FUNCTION_BLOCK PUBLIC LotLogging
VAR_INPUT
END_VAR
VAR_OUTPUT
END_VAR
VAR
	PrevLotInProgress : BOOL;
	TimeToLogLot : TON;
END_VAR

IF (NOT LotsData.Lot.LotInProgress) AND PrevLotInProgress THEN
	// create a lot report here and store it
	P_TextModeWriteLot.WriteData := TRUE;	   
END_IF
PrevLotInProgress := LotsData.Lot.LotInProgress;

END_FUNCTION_BLOCK

(* stored: Version 1.1.0.1, ProductVersion 3.1.4020.12
   POU LotLogging: Id {5cf7cc70-e7e4-43f5-9ece-da902bcdcb94}, SpecialFunc None *)
